FUNCTION_BLOCK EcMasterGetDeviceCRC IMPLEMENTS IEcTask
VAR_INPUT
END_VAR
VAR_OUTPUT
END_VAR
VAR
	iState : INT;
	getDeviceCRC : Tc2_EtherCAT.FB_EcGetSlaveCrcErrorEx;
	_execute: BOOL;
	_done: BOOL;
	_busy: BOOL;
	_error: BOOL;
	_netId: AMSNETID;
END_VAR

CASE iState OF
	0:
		IF _execute THEN
			_done := FALSE;
			_busy := TRUE;
			_error := FALSE;
			getDeviceCRC.bExecute := TRUE;
			IF getDeviceCRC.bBusy THEN
				iState := 10;
				_execute := false;
			END_IF
		END_IF
	10:
		IF NOT getDeviceCRC.bBusy THEN
			IF NOT getDeviceCRC.bError THEN
				_done := TRUE;
			ELSE
				_error := TRUE;
			END_IF
			_busy := FALSE;
			getDeviceCRC.bExecute := FALSE;
			iState := 0;
		END_IF
END_CASE

getDeviceCRC(sNetId := Tc2_System.F_CreateAmsNetId(nIds := NetId));

{warning 'add method implementation '}
METHOD Abort : BOOL
getDeviceCRC.bExecute := FALSE;
_busy := FALSE;
_execute := FALSE;
Abort := TRUE;
iState := 0;
END_METHOD

{warning 'add property implementation'}
PROPERTY Busy : BOOL
GET
Busy := _busy;
END_GET
END_PROPERTY

PROPERTY DeviceAddr : uint
GET
DeviceAddr := getDeviceCRC.nSlaveAddr;
END_GET
SET
getDeviceCRC.nSlaveAddr := DeviceAddr;
END_SET
END_PROPERTY

PROPERTY DeviceCRC :  ST_EcCrcErrorEx
GET
DeviceCRC := getDeviceCRC.crcError;
END_GET
END_PROPERTY

{warning 'add property implementation'}
PROPERTY Done : BOOL
GET
Done := _done;
END_GET
END_PROPERTY

{warning 'add property implementation'}
PROPERTY Error : BOOL
GET
Error := _error;
END_GET
END_PROPERTY

{warning 'add method implementation '}
METHOD Execute : BOOL
IF NOT getDeviceCRC.bBusy THEN
	Execute := _execute := true;
END_IF
END_METHOD

{warning 'add property implementation'}
PROPERTY NetID : amsnetid
GET
NetID := _netId;
END_GET
SET
_netId := NetID;
END_SET
END_PROPERTY

END_FUNCTION_BLOCK

(* stored: Version 1.1.0.1, ProductVersion 3.1.4024.11
   POU EcMasterGetDeviceCRC: Id {acf0f775-e600-43e4-8f7e-1fecde418fdc}, SpecialFunc None
   Method Abort: Id {7a77e909-7b5e-48c6-91f9-3baff34dc81d}
   Property Busy: Id {69665580-7eb3-4846-9f28-8225ce1cbd4f}
   Get Get: Id {79dac96c-22eb-48c0-9b19-61b51cbd9283}
   Property DeviceAddr: Id {0df72374-07d3-481f-a188-14bd0c254ca9}
   Get Get: Id {a3fac021-c983-445c-bd41-8d001103a5ac}
   Set Set: Id {d45648f4-5fab-4540-8366-4fe85384c617}
   Property DeviceCRC: Id {19557706-231a-4a3b-b8bc-e2f3dc29c070}
   Get Get: Id {e3792a99-24b9-46e1-a2b8-a779c9c0aff6}
   Property Done: Id {71014689-839c-4777-8e1a-b2aa422bee9e}
   Get Get: Id {79521043-885b-408f-8db2-1d3df7f55af6}
   Property Error: Id {47342163-b180-4fab-b181-f062d32dc03f}
   Get Get: Id {d2b48224-ee5e-4663-8d72-fdece8ca326c}
   Method Execute: Id {a5777f9d-1ed9-4ac2-bcc9-405887e9d033}
   Property NetID: Id {04038629-ac9f-4249-b71d-86888cacb94b}
   Get Get: Id {152ff8db-6e3e-4101-ae9d-ebf7c4a251db}
   Set Set: Id {9e5bbebc-ded7-47e8-abb6-414defa8f4f5} *)
